VAR_GLOBAL PERSISTENT 
	
ATL:ATL;

END_VAR

(* stored: Version 1.1.0.1, ProductVersion 3.1.4024.9
   GVL _PE: Id {82cc4c82-2a76-4751-92b7-08ad0e41a9d0} *)
